PROGRAM HMI
VAR

//OpenDialog:FbOpenDialog;
END_VAR

END_PROGRAM

(* stored: Version 1.1.0.1, ProductVersion 3.1.4024.12
   POU HMI: Id {69636261-3123-453c-af0c-f3ab55ea0690}, SpecialFunc None *)
